Fanuc KAREL source: kf00104.KL

-- PROVISIONAL review KL for V1013-1; original PC SHA256 be90d4fb7c3b8e42a701b321801147602c7f8b7f89694001abc2816b4952897b
-- Incomplete behavior may be omitted. Consult companion uncertainty JSON. Do not deploy.
PROGRAM KF00104
%NOLOCKGROUP
BEGIN
  -- UNRESOLVED_PC offsets 5-16; opcodes 2E,23
  -- UNRESOLVED_PC offsets 21-32; opcodes 2E,23
  -- UNRESOLVED_PC offsets 37-57; opcodes 27,27,9D,22,2A,22,31
  -- UNRESOLVED_PC offsets 62-66; opcodes 7F
END KF00104
